// TIA Portal V17 export
TagTable "Codex_Popup_Sim_Int_Tags"
  Sim_SelectedCompID : Int  (1 s, start 1)   // Popup simulation selected component ID.
